FUNCTION_BLOCK ABSTRACT DistanceSensorBase EXTENDS TExecution IMPLEMENTS IDevice
VAR_INPUT
END_VAR
VAR_OUTPUT
END_VAR
VAR
	{attribute 'OPC.UA.DA' := '0'}
	_name : STRING;
	{attribute 'OPC.UA.DA' := '0'}
	_deviceID : STRING;					
	{attribute 'OPC.UA.DA' := '0'}
	_family : DeviceFamily;	
	{attribute 'OPC.UA.DA' := '0'}
	_logger : Logger;
	{attribute 'OPC.UA.DA' := '0'}
	_message : StringBuilder;
	{attribute 'OPC.UA.DA' := '0'}
	_distanceSensorConfig : DeviceConfiguration;
END_VAR

PROPERTY DeviceID : STRING
GET
DeviceID := _deviceID;
END_GET
SET
_deviceID := DeviceID;
END_SET
END_PROPERTY

PROPERTY Family : DeviceFamily
GET
Family := _family;
END_GET
SET
_family := Family;
END_SET
END_PROPERTY

PROPERTY Name : STRING
GET
Name := _name;
END_GET
SET
_name := Name;
END_SET
END_PROPERTY

END_FUNCTION_BLOCK

(* stored: Version 1.1.0.1, ProductVersion 3.1.4024.3
   POU DistanceSensorBase: Id {c210bc83-a234-4906-b394-015f9aa20866}, SpecialFunc None
   Property DeviceID: Id {f52b8b85-7fc0-4b7b-9447-a31dae20fd59}
   Get Get: Id {a986bcda-cfc9-471d-a243-b301336ba57c}
   Set Set: Id {46eccb5a-5471-4e3d-8e8c-35ede67c4ea7}
   Property Family: Id {708e9eaa-d62e-4b80-848d-e12438309e0d}
   Get Get: Id {cba97d0c-fdb2-4dd8-9e33-39d28b22ccd1}
   Set Set: Id {143f6daf-0bad-4ae8-a639-3beda2d86efc}
   Property Name: Id {0a802fc8-4d27-4245-a042-86fff028a584}
   Get Get: Id {33715da5-a9e4-4b80-89df-0196f20fd49e}
   Set Set: Id {e5623566-1b1d-4791-8172-2c00cf23b0b0} *)
